{attribute 'qualified_only'}
{attribute 'strict'}
TYPE AlarmPriority :
(
	A := 0, B, C
);
END_TYPE

(* stored: Version 1.1.0.1, ProductVersion 3.1.4024.6
   DUT AlarmPriority: Id {7fbc5980-8de2-4d6c-a904-4af25c47065e} *)
